PROGRAM POU
VAR
	Paso: INT;
	SALTO_A_30: BOOL;
	SALTO_A_10: BOOL;	
	SALTO_A_20: BOOL;	

	Trans0: BOOL;
	VarOut AT %Q*: BOOL;
	VarIn AT %I*: BOOL;
	VarOut2 AT %Q*: BOOL;
	VarIn2 AT %I*: BOOL;
END_VAR

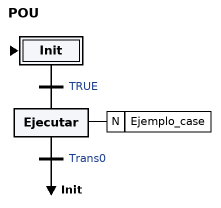
INITIAL_STEP Init:
END_STEP
TRANSITION FROM Init TO Ejecutar
    := TRUE;
END_TRANSITION
STEP Ejecutar:
    Ejemplo_case(N);
END_STEP
TRANSITION FROM Ejecutar TO Init
    := Trans0;
END_TRANSITION

ACTION Ejemplo_case:
     ADSLOGDINT(msgCtrlMask:= ADSLOG_MSGTYPE_LOG, msgFmtStr := 'Paso Actual: %d', dintArg := Paso);

CASE Paso OF
	10:
     ADSLOGSTR(msgCtrlMask:= ADSLOG_MSGTYPE_LOG, msgFmtStr := 'EN PASO 10' , strArg := ' '); 
     Paso := 20;
	
	20:
	
	 IF SALTO_A_30 THEN
		 ADSLOGSTR(msgCtrlMask:= ADSLOG_MSGTYPE_LOG, msgFmtStr := 'SALTO A 30' , strArg := ' ');
		 Paso := 30;
	 END_IF
	  IF SALTO_A_10 THEN
		 ADSLOGSTR(msgCtrlMask:= ADSLOG_MSGTYPE_LOG, msgFmtStr := 'SALTO A 10' , strArg := ' ');
		 Paso := 10;
	  ELSE
	      ADSLOGSTR(msgCtrlMask:= ADSLOG_MSGTYPE_LOG, msgFmtStr := 'ELSE PASO 20' , strArg := ' ');
		  END_IF
		   
	30:
	     ADSLOGSTR(msgCtrlMask:= ADSLOG_MSGTYPE_LOG, msgFmtStr := 'EN PASO 30' , strArg := ' ');
          IF SALTO_A_20 THEN
		 ADSLOGSTR(msgCtrlMask:= ADSLOG_MSGTYPE_LOG, msgFmtStr := 'SALTO A 30' , strArg := ' ');
		 Paso := 20;
		 END_IF

END_CASE
END_ACTION

END_PROGRAM

(* stored: Version 1.1.0.1, ProductVersion 3.1.4024.12
   POU POU: Id {87c77caa-00c7-42a1-a3fd-614363e47b75}, SpecialFunc None
   Action Ejemplo_case: Id {ec0d25cc-5d85-4ff2-b011-e10732849df1} *)
